# EPICS StreamDevice protocol: iocBoot/iocdcu/dcu.proto
Terminator = CR;

getstream {
  in "%s";
  }
